{attribute 'linkalways'} 
{attribute 'no_explicit_call' := 'This FB is a CLASS and must be accessed using methods or properties'}
{attribute 'enable_dynamic_creation'}
FUNCTION_BLOCK Node_F_VN_MatchContours1vsN EXTENDS VisionNode
VAR
    ipRefContour : _ITcVnContainer;
    ipContours : _ITcVnContainer;
    ipMatchIndexes : _ITcVnContainer;
    ipDissimilarities : _ITcVnContainer;
    fDissimilarityThreshold : _LREAL(0.0);
    eComparisonMethod : _ETcVnContoursMatchComparisonMethod(ETcVnContoursMatchComparisonMethod.TCVN_CMCM_CONTOURS_MATCH_I1);
    hrPrev : _HRESULT(S_OK);
	hresult : _HRESULT(S_OK);
END_VAR

METHOD PUBLIC  Clone : I_Node
VAR
	pNode : POINTER TO Node_F_VN_MatchContours1vsN;
END_VAR
pNode := __NEW(Node_F_VN_MatchContours1vsN);
Clone := pNode^;
END_METHOD

METHOD FB_init : BOOL
VAR_INPUT
	bInitRetains : BOOL; // if TRUE, the retain variables are initialized (warm start / cold start)
	bInCopyCode : BOOL;  // if TRUE, the instance afterwards gets moved into the copy code (online change)
END_VAR
AddInput('ipRefContour', ipRefContour);
AddInput('ipContours', ipContours);
AddParameter('fDissimilarityThreshold', fDissimilarityThreshold);
AddParameter('eComparisonMethod', eComparisonMethod);
AddInput('hrPrev', hrPrev);
AddOutput('ipMatchIndexes', ipMatchIndexes);
AddOutput('ipDissimilarities', ipDissimilarities);
AddOutput('hresult', hresult);
END_METHOD

METHOD PROTECTED OnExecute
hresult.Value := F_VN_MatchContours1vsN(
	ipRefContour := ipRefContour.Value,
    ipContours := ipContours.Value,
    ipMatchIndexes := ipMatchIndexes.Value,
    ipDissimilarities := ipDissimilarities.Value,
    fDissimilarityThreshold := fDissimilarityThreshold.Value,
    eComparisonMethod := eComparisonMethod.Value,
	hrPrev:= hrPrev.Value);
END_METHOD

METHOD PUBLIC PreExecutionCheck
VAR_INPUT
	Check : I_PreExecutionChecks;
END_VAR
Check.IsTrue(ipRefContour.IsValid, 'ipRefContour must be a valid container');
Check.IsTrue((ipRefContour.IsType(TC_GLOBAL_CONST_LIST.ContainerType_Vector_TcVnPoint2_DINT) OR
              ipRefContour.IsType(TC_GLOBAL_CONST_LIST.ContainerType_Vector_TcVnPoint2_REAL)),
              'ipRefContour contains incorrect type');
              
Check.IsTrue(ipContours.IsValid, 'ipContours must be a valid container');
Check.IsTrue(ipContours.IsType(TC_GLOBAL_CONST_LIST.ContainerType_Vector_Vector_TcVnPoint2_DINT), 'ipContours contains incorrect type');
END_METHOD

END_FUNCTION_BLOCK

(* stored: Version 1.1.0.1, ProductVersion 3.1.4026.13
   POU Node_F_VN_MatchContours1vsN: Id {f3ef6208-78d6-07b9-3917-8d8e26161702}, SpecialFunc None
   Folder Constructor: Id {1ad2ebe5-8952-0915-22d2-98082ea4b003}
   Method Clone: Id {fadcc0e3-aa9b-0ac7-1570-4cb216782200}
   Method FB_init: Id {e53eef33-44b6-0232-0b97-c66af5716025}
   Method OnExecute: Id {56ea18f8-48e0-0d72-322a-0f299c579b93}
   Method PreExecutionCheck: Id {c8afdda7-003a-062b-237f-dadf1349e3a2} *)
